// TIA Portal V15.1 export
// export: Created 2024-06-21T08:41:11.5560262Z, ExportSetting WithDefaults, DisplayName Totally Integrated Automation Portal, DisplayVersion V15.1 Update 5, DisplayName TIA Portal Openness, DisplayVersion V15.1 Update 5, DisplayName SINAMICS Startdrive Advanced, DisplayVersion V15.1, DisplayName G130, G150, S120, S150, SINAMICS MV, S210, DisplayVersion V15.1, DisplayName G110M, G120, G120C, G120D, G120P, DisplayVersion V15.1, DisplayName STEP 7 Professional, DisplayVersion V15.1 Update 5, DisplayName STEP 7 Safety, DisplayVersion V15.1, DisplayName WinCC Professional, DisplayVersion V15.1 Update 5, DisplayName SIMATIC Visualization Architect, DisplayVersion V15.1
FUNCTION "LGBRdWrRecipe" : Void   // FC6614, SCL
{ S7_Optimized_Access := 'TRUE' }
VERSION : 0.1
// stored: AutoNumber false, IsIECCheckEnabled false, SetENOAutomatically False, UDAEnableTagReadback false
   VAR_INPUT
      I_Index : Int;
      I_EnableWrite : Bool;
      I_EnableRead : Bool;
   END_VAR
   VAR_IN_OUT
      IO_Done : Bool;
      IO_Recipe : Array[1..35] of "TCRecipe";
      IO_RecipeData : "TCRecipe";
   END_VAR
   VAR_TEMP
      RetVal : Int;
   END_VAR
BEGIN
   //------------------------------------------------------------------------------------------------
   //Handles the  writing of the data to the recipe 
   //------------------------------------------------------------------------------------------------

   //------------------------------------------------------------------------------------------------
   //Check change of input indexes and if true >>> write data to 
   //------------------------------------------------------------------------------------------------
   IF #I_EnableWrite = true THEN

       #IO_RecipeData := #IO_Recipe[#I_Index];
       #IO_Done := true;

   END_IF;

   IF #I_EnableRead = true AND #IO_RecipeData.RecipeLineStart = #I_Index THEN
       #IO_Recipe[#I_Index] := #IO_RecipeData;
       #IO_Done := true;

   END_IF;
END_FUNCTION
